FUNCTION_BLOCK FB_StatesAndModes
VAR_INPUT
END_VAR
VAR_OUTPUT
END_VAR
VAR
END_VAR

END_FUNCTION_BLOCK

(* stored: Version 1.1.0.1
   POU FB_StatesAndModes: Id {6f344e3b-9128-4c83-8a29-98893305b6bf}, SpecialFunc None *)
